FUNCTION_BLOCK CROSSCOMM_SENDER_5766F27C0FBCC110 (* Service Interface Function Block Type *)
  (* Standard: 61499-2 *)
  (* Version 0.0, 9/22/2017, bababen, nxtControl GmbH, template *)
  PACKAGE Main;
  (* Compiler Cpp nxtControl builtin 1.0 *)
  {SET_ATTRIBUTE(Runtime.FBType.ImplementingType, Runtime.System#DYNGEN_CROSSCOMM_SENDER)}
  {SET_ATTRIBUTE(Configuration.GenericFBType.InterfaceParams, Runtime.System#<InterfaceList> <EventInputs> <Event Name="INITO" /> <Event Name="CNF"> <With Var="RetractLift" /> <With Var="ExtendLift" /> </Event> </EventInputs> <InputVars> <VarDeclaration Name="RetractLift" Type="BOOL" /> <VarDeclaration Name="ExtendLift" Type="BOOL" /> </InputVars> </InterfaceList>)}
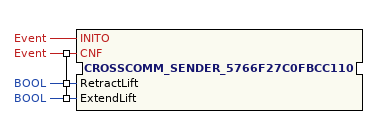
  EVENT_INPUT
    INITO;
    CNF WITH RetractLift, ExtendLift;
  END_EVENT
  VAR_INPUT
    RetractLift : BOOL;
    ExtendLift : BOOL;
  END_VAR
  EC_STATES
    START;
  END_STATES
END_FUNCTION_BLOCK
